{attribute 'GeneratedUsingTerminal: EK1100-0000-0018'}
{attribute addProperty BoxType "EK1100-0000-0018"}
{attribute addProperty Id "Beckhoff_EL73xxEK1122Beckhoff_EL73xxEK1122_3D63295F2A_0001_EL7332_0000_0016EL7332_5D0CE0D446A_0002_EL7332_0000_0017EL7332_5D0CE0D446A_0003_EL7332_0000_0018EL7332_5D0CE0D446A_0004_EL7332_0000_0019EL7332_5D0CE0D446A_0005_EL7332_0000_0020EL7332_5D0CE0D446A_0006_EL7332_0000_0021EL7332_5D0CE0D446A_0007_EL7332_0000_0022EL7332_5D0CE0D446A_0008_EL7332_0000_0023EL7332_5D0CE0D446A_0009_EL7332_0000_0024EL7332_5D0CE0D446A_0010_EL7342_0000_0016EL7342_2F848FE386A_0011_EL7342_0000_0017EL7342_2F848FE386A_0012_EL7342_0000_0018EL7342_2F848FE386A_0013_EL7342_0000_0019EL7342_2F848FE386A_0014_EL7342_0000_0020EL7342_2F848FE386A_0015_EL7342_0000_0021EL7342_2F848FE386A_0016_EL7342_0000_0022EL7342_2F848FE386A_0017_EL7342_0000_0023EL7342_A882861088A_0018_EL7342_0035_0019EL7342_2F848FE386A_0019_EL7342_0035_0020EL7342_2F848FE386"}
{attribute addProperty CRC "2225528602"}
{attribute addProperty Size "1278"}
TYPE Beckhoff_EL73xx_84A6DF1A EXTENDS EK1100_AB5A9467 :
STRUCT
	{attribute addProperty Name "Beckhoff_EL73xxEK1122"}
	Beckhoff_EL73xxEK1122 : Beckhoff_EL73xxEK1122_3D63295F;
	{attribute addProperty Name "A_0001_EL7332_0000_0016"}
	A_0001_EL7332_0000_0016 : EL7332_5D0CE0D4;
	{attribute addProperty Name "A_0002_EL7332_0000_0017"}
	A_0002_EL7332_0000_0017 : EL7332_5D0CE0D4;
	{attribute addProperty Name "A_0003_EL7332_0000_0018"}
	A_0003_EL7332_0000_0018 : EL7332_5D0CE0D4;
	{attribute addProperty Name "A_0004_EL7332_0000_0019"}
	A_0004_EL7332_0000_0019 : EL7332_5D0CE0D4;
	{attribute addProperty Name "A_0005_EL7332_0000_0020"}
	A_0005_EL7332_0000_0020 : EL7332_5D0CE0D4;
	{attribute addProperty Name "A_0006_EL7332_0000_0021"}
	A_0006_EL7332_0000_0021 : EL7332_5D0CE0D4;
	{attribute addProperty Name "A_0007_EL7332_0000_0022"}
	A_0007_EL7332_0000_0022 : EL7332_5D0CE0D4;
	{attribute addProperty Name "A_0008_EL7332_0000_0023"}
	A_0008_EL7332_0000_0023 : EL7332_5D0CE0D4;
	{attribute addProperty Name "A_0009_EL7332_0000_0024"}
	A_0009_EL7332_0000_0024 : EL7332_5D0CE0D4;
	{attribute addProperty Name "A_0010_EL7342_0000_0016"}
	A_0010_EL7342_0000_0016 : EL7342_2F848FE3;
	{attribute addProperty Name "A_0011_EL7342_0000_0017"}
	A_0011_EL7342_0000_0017 : EL7342_2F848FE3;
	{attribute addProperty Name "A_0012_EL7342_0000_0018"}
	A_0012_EL7342_0000_0018 : EL7342_2F848FE3;
	{attribute addProperty Name "A_0013_EL7342_0000_0019"}
	A_0013_EL7342_0000_0019 : EL7342_2F848FE3;
	{attribute addProperty Name "A_0014_EL7342_0000_0020"}
	A_0014_EL7342_0000_0020 : EL7342_2F848FE3;
	{attribute addProperty Name "A_0015_EL7342_0000_0021"}
	A_0015_EL7342_0000_0021 : EL7342_2F848FE3;
	{attribute addProperty Name "A_0016_EL7342_0000_0022"}
	A_0016_EL7342_0000_0022 : EL7342_2F848FE3;
	{attribute addProperty Name "A_0017_EL7342_0000_0023"}
	A_0017_EL7342_0000_0023 : EL7342_A8828610;
	{attribute addProperty Name "A_0018_EL7342_0035_0019"}
	A_0018_EL7342_0035_0019 : EL7342_2F848FE3;
	{attribute addProperty Name "A_0019_EL7342_0035_0020"}
	A_0019_EL7342_0035_0020 : EL7342_2F848FE3;
END_STRUCT
END_TYPE

(* stored: Version 1.2.0.0, ProductVersion 3.1.4024.9
   DUT Beckhoff_EL73xx_84A6DF1A: Id {ee6ce379-84d2-4cb1-944f-f922fe19aaad} *)
